{attribute 'qualified_only'}
VAR_GLOBAL PERSISTENT 
	Status :ARRAY[1..MM_CONST.MAX_VEHICLES] OF PartDataType;
END_VAR

(* stored: Version 1.1.0.1, ProductVersion 3.1.4020.12
   GVL PartsData: Id {24ca4289-9a4a-4961-a2cc-e5d0f97296fb} *)
